PROGRAM POU
VAR
END_VAR

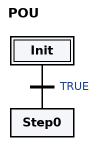
INITIAL_STEP Init:
END_STEP
TRANSITION FROM Init TO Step0
    := TRUE;
END_TRANSITION
STEP Step0:
END_STEP

END_PROGRAM

(* stored: Version 1.1.0.1, ProductVersion 3.1.4024.12
   POU POU: Id {e16536b7-1c0b-4946-baaf-851eba1556f6}, SpecialFunc None *)
